// LS Electric XG5000 project: 신호등
// PLC LSPLC
// module base 0 slot 0: 입출력 모듈:XBC-DR14E (DC 24V 입력 8점, 릴레이 출력 6점)

PROGRAM NewProgram (task: 스캔 프로그램)

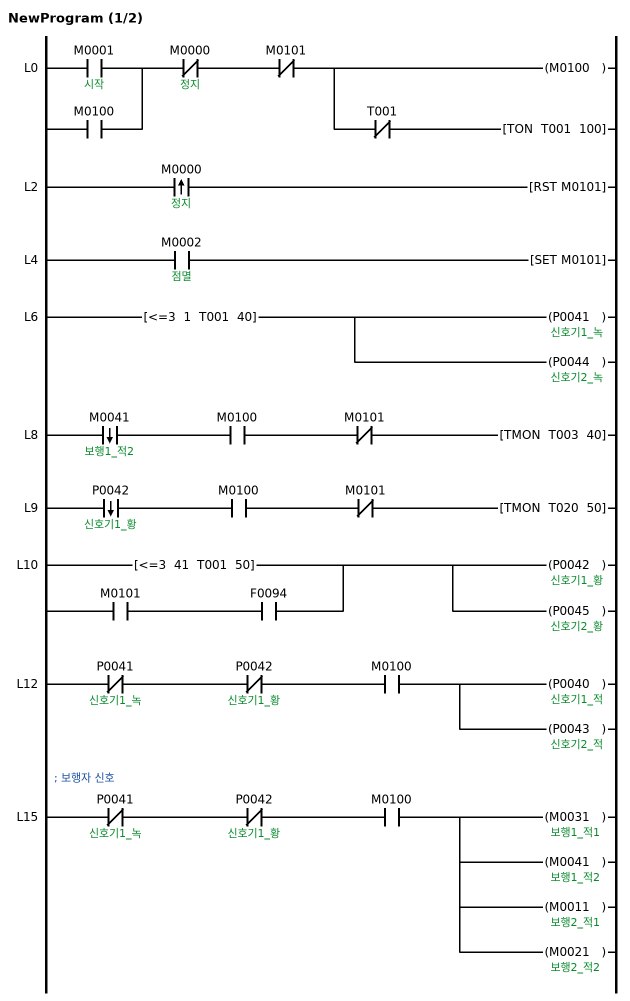
; L0
LOAD      M0001	// 시작
OR        M0100
AND NOT   M0000	// 정지
AND NOT   M0101
OUT       M0100
AND NOT   T001
TON       T001 100
; L2
LOADP     M0000	// 정지
RST       M0101
; L4
LOAD      M0002	// 점멸
SET       M0101
; L6
LOAD<=3   1 T001 40
OUT       P0041	// 신호기1_녹
OUT       P0044	// 신호기2_녹
; L8
LOADN     M0041	// 보행1_적2
AND       M0100
AND NOT   M0101
TMON      T003 40
; L9
LOADN     P0042	// 신호기1_황
AND       M0100
AND NOT   M0101
TMON      T020 50
; L10
LOAD<=3   41 T001 50
LOAD      M0101
AND       F0094
OR LOAD
OUT       P0042	// 신호기1_황
OUT       P0045	// 신호기2_황
; L12
LOAD NOT  P0041	// 신호기1_녹
AND NOT   P0042	// 신호기1_황
AND       M0100
OUT       P0040	// 신호기1_적
OUT       P0043	// 신호기2_적
// 보행자 신호
; L15
LOAD NOT  P0041	// 신호기1_녹
AND NOT   P0042	// 신호기1_황
AND       M0100
OUT       M0031	// 보행1_적1
OUT       M0041	// 보행1_적2
OUT       M0011	// 보행2_적1
OUT       M0021	// 보행2_적2

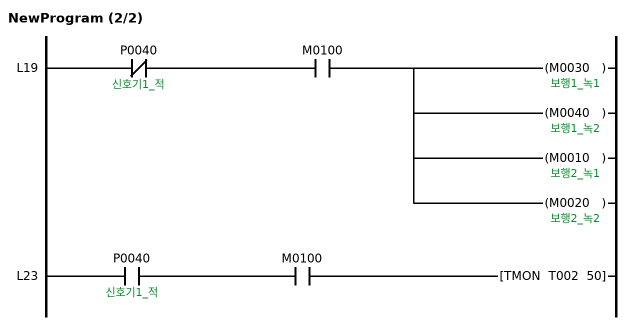
; L19
LOAD NOT  P0040	// 신호기1_적
AND       M0100
OUT       M0030	// 보행1_녹1
OUT       M0040	// 보행1_녹2
OUT       M0010	// 보행2_녹1
OUT       M0020	// 보행2_녹2
; L23
LOAD      P0040	// 신호기1_적
AND       M0100
TMON      T002 50